INTERFACE I_CleanDevice

METHOD mAbort : BOOL
VAR_INPUT
END_VAR
END_METHOD

METHOD mAckError
VAR_INPUT
END_VAR
END_METHOD

METHOD mOperation : BOOL
VAR_INPUT
	iI_Step : INT;
END_VAR
END_METHOD

METHOD mSetMode : BOOL
VAR_INPUT
	sI_CleanMode : EN_CLEANING_OP;
END_VAR
END_METHOD

PROPERTY sStatus : ST_CLEANING_DEV_STATUS
GET
END_GET
END_PROPERTY

END_INTERFACE

(* stored: Version 1.1.0.1, ProductVersion 3.1.4024.11
   Itf I_CleanDevice: Id {f9467c5b-d9bf-4936-be7b-12ebef9b078d}
   Method mAbort: Id {721a87b1-409e-499c-b73e-95b1299e1770}
   Method mAckError: Id {8150d4da-4956-4062-a8af-28026f6eb0ff}
   Method mOperation: Id {fc55badb-54e3-4dd7-b7bb-c79540edd7f8}
   Method mSetMode: Id {cda35f5b-2fed-46c8-a615-45fa3f48223c}
   Property sStatus: Id {67f9f641-6e10-4815-99f2-46d9edead7bb}
   Get Get: Id {aeefb536-a171-43d4-9d92-b487c509c71b} *)
